ABB RobotStudio station: Estacion_Proyecto.rspag

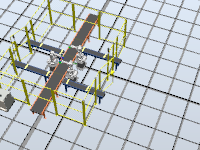
--- station ---
Station Estacion_Proyecto (saved by RobotStudio 20.4.9280.0)
Controller Controlador_Vajilla, task T_ROB3: task frame (RAPID world) sits at (0, 0, 0) mm in the station
Controller Controlador_Vajilla, task T_ROB2: task frame (RAPID world) sits at (0, 0, 0) mm in the station
Controller Controlador_Vajilla, task T_ROB1: task frame (RAPID world) sits at (0, 0, 0) mm in the station
Controller Controlador_Vajilla
  mechanical unit ROB_1: IRB140_6_81_C_03_1, 6 joints, base frame (0, 570, 550) mm, rotated rx 0 ry 0 rz -90 deg
  mechanical unit ROB_2: IRB140_6_81_C_03_2, 6 joints, base frame (1000, 555, 550) mm, rotated rx 0 ry 0 rz -90 deg
  mechanical unit ROB_3: IRB140_6_81_C_03_3, 6 joints, base frame (732.5, -570, 550) mm, rotated rx 0 ry 0 rz 90 deg
Layout (positions relative to the parent item):
  - IRB140_6_81_C_03_1 [mechanism, from Robots\IRB140_6_81_C_G_03.rslib] at (0, 570, 550) mm, rotated rx 0 ry 0 rz -90 deg; joint values [0, 0, 0, 0, 0.5236, 0] (rad or m)
  - IRB140_6_81_C_03_2 [mechanism, from Robots\IRB140_6_81_C_G_03.rslib] at (1000, 555, 550) mm, rotated rx 0 ry 0 rz -90 deg; joint values [0, -0.0417, 0.0409, 0, 0.5244, 0] (rad or m)
  - IRB140_6_81_C_03_3 [mechanism, from Robots\IRB140_6_81_C_G_03.rslib] at (732.5, -570, 550) mm, rotated rx 0 ry 0 rz 90 deg; joint values [0, 0, 0, 0, 0.5236, 0] (rad or m)
  - Sockel_IRB140_500mm_3 [part, from Proyecto\53244bc2-0fdb-48b8-abaf-b031e49cfeeesockel_irb140_500mm.rslib] at (732.5, -570, 0) mm, rotated rx 0 ry 0 rz 90 deg
  - Sockel_IRB140_500mm_1 [part, from Proyecto\53244bc2-0fdb-48b8-abaf-b031e49cfeeesockel_irb140_500mm.rslib] at (0, 570, 0) mm, rotated rx 0 ry 0 rz -90 deg
  - Sockel_IRB140_500mm_2 [part, from Proyecto\53244bc2-0fdb-48b8-abaf-b031e49cfeeesockel_irb140_500mm.rslib] at (1000, 555, 0) mm, rotated rx 0 ry 0 rz -90 deg
  - Linea_Plato_Pando [part] at (-250, 0, 0) mm
  - Linea_Plato_Postre [part] at (0, -6.06, 0) mm
  - Linea_Plato_Hondo [part]
  - Linea_Vaso [part]
  - VacuumToolCreator [smart component, from Proyecto\d28571e4-d633-4a15-b430-832653a4066fvacuumtoolcreator.rslib]
      properties: Tool Name=VacuumTool; TCP Name=tVacuum; TCP Position=[0 0 0.049]; TCP Orientation=[0 0 0]; Flange Diameter=0.055; Length=0.1; Width=0.1; Solids only=false; GeneratedTool=VacuumTool
  - VacuumTool [mechanism, from modelados\VacuumTool.rslib] at (0, 63.71, 1229.5) mm, rotated rx 180 ry 60 rz 90 deg
  - Conveyor_PH [smart component]
      signals: DO ACR, DI ACV, DI DCV, DI INC
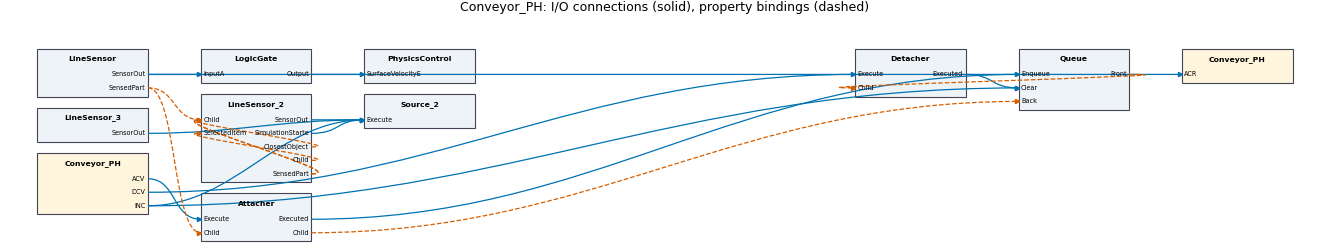
      connections:
        LineSensor.SensorOut -> LogicGate.InputA
        LogicGate.Output -> PhysicsControl.SurfaceVelocityEnabled
        LineSensor_2.SensorOut -> Source_2.Execute
        LineSensor_3.SensorOut -> Source_2.Execute
        SimulationEvents.SimulationStarted -> Source_2.Execute
        LineSensor.SensorOut -> Conveyor_PH.ACR
        Conveyor_PH.ACV -> Attacher.Execute
        Attacher.Executed -> Queue.Enqueue
        Detacher.Executed -> Queue.Clear
        Conveyor_PH.DCV -> Detacher.Execute
        Conveyor_PH.INC -> Source_2.Execute
        Conveyor_PH.INC -> Queue.Clear
        LineSensor.SensedPart => Attacher.Child
        ClosestObject.ClosestObject => Detacher.Child
        Attacher.Child => DataTable.SelectedItem
        VolumeSensor.SensedPart => Detacher.Child
        LineSensor_5.SensedPart => Detacher.Child
        LineSensor.SensedPart => Attacher.Child
        Attacher.Child => Queue.Back
        Queue.Front => Detacher.Child
    - Source_2 [smart component, from Components\Source.rslib] at (159.05, -900.89, 1238.71) mm, rotated rx -56.63 ry -24.63 rz -15.35 deg
        properties: Source=plato_hondo; Copy=(none); Parent=(none); Position=[-0.55 2.2 0.6]; Orientation=[0 0 0]; Transient=true; PhysicsBehavior=3
    - LineSensor [smart component, from Components\LineSensor.rslib]
        properties: Start=[-0.4 0.47 0.6405]; End=[-0.7 0.47 0.6405]; Radius=0.004; SensedPart=(none); SensedPoint=[0 0 0]
      - _sensorPart_ [part]
    - PhysicsControl [smart component, from Components\PhysicsControl.rslib] at (0, -15, 0) mm
        properties: Object=Linea_Plato_Hondo; Behavior=1; SurfaceVelocity=0.3302
    - LogicGate [smart component, from Components\LogicGate.rslib]
        properties: Operator=NOT; Delay=0
    - LineSensor_3 [smart component, from Components\LineSensor.rslib]
        properties: Start=[-0.4 1.6 0.6405]; End=[-0.7 1.6 0.6405]; Radius=0.004; SensedPart=(none); SensedPoint=[0 0 0]
      - _sensorPart_ [part]
    - Attacher [smart component, from Components\Attacher.rslib]
        properties: Parent=VacuumTool; Flange=0; Child=(none); Mount=false; Offset=[0 0 0]; Orientation=[0 0 0]
    - Queue [smart component, from Components\Queue.rslib]
        properties: Back=(none); Front=(none); Queue=; NumberOfObjects=0
    - Detacher [smart component, from Components\Detacher.rslib]
        properties: Child=(none); KeepPosition=true
  - Conveyor_Principal [smart component]
      signals: DI INC, DI MOV, DO ACR_1P, DO ACR_3P
      connections:
        Conveyor_Principal.INC -> Source.Execute
        Conveyor_Principal.MOV -> LogicGate_2.InputA
        LogicGate.Output -> LogicGate_2.InputB
        LogicGate_2.Output -> PhysicsControl.SurfaceVelocityEnabled
        PlaneSensor.SensorOut -> LogicGate.InputA
        PlaneSensor.SensorOut -> Conveyor_Principal.ACR_1P
        PlaneSensor_2.SensorOut -> Conveyor_Principal.ACR_3P
        PlaneSensor_3.SensorOut -> Source.Execute
    - PhysicsControl [smart component, from Components\PhysicsControl.rslib]
        properties: Object=Linea_Principal; Behavior=1; SurfaceVelocity=0.3
    - Source [smart component, from Components\Source.rslib] at (-3.56, 0, 724.94) mm
        properties: Source=caja; Copy=(none); Parent=(none); Position=[-2.5 0 0.6]; Orientation=[0 0 3.14159265358979]; Transient=true; PhysicsBehavior=3
    - LogicGate [smart component, from Components\LogicGate.rslib]
        properties: Operator=NOT; Delay=0
    - LogicGate_2 [smart component, from Components\LogicGate.rslib]
        properties: Operator=OR; Delay=0
    - PlaneSensor [smart component, from Components\PlaneSensor.rslib]
        properties: Origin=[0.12 -0.3 0.605]; Axis1=[0 0.6 0]; Axis2=[0 0 0.1]; SensedPart=(none)
      - _sensorPart_ [part]
    - PlaneSensor_2 [smart component, from Components\PlaneSensor.rslib]
        properties: Origin=[1.3 -0.26 0.605]; Axis1=[-0.00064 0.52 0]; Axis2=[0 0 0.1]; SensedPart=(none)
      - _sensorPart_ [part]
    - PlaneSensor_3 [smart component, from Components\PlaneSensor.rslib]
        properties: Origin=[-1.03 -0.3 0.601]; Axis1=[3E-06 0.6 0]; Axis2=[0 0 0.1]; SensedPart=(none)
      - _sensorPart_ [part]
  - Conveyor_PP [smart component]
      signals: DI ACV_3, DI DCV_3, DI INC_3, DO ACR_3
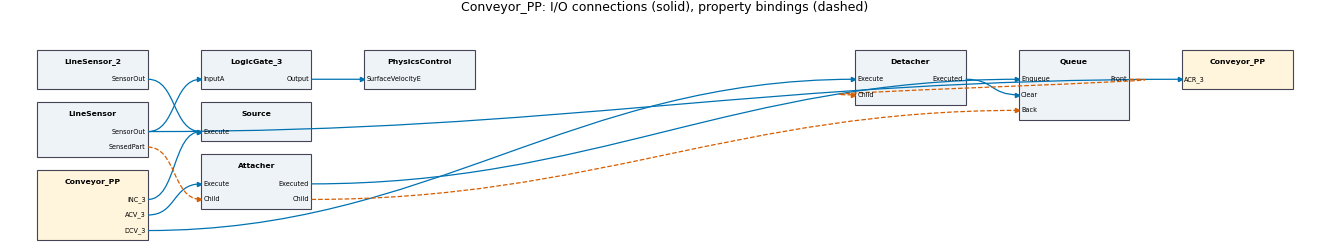
      connections:
        LineSensor_2.SensorOut -> Source.Execute
        LineSensor.SensorOut -> LogicGate_3.InputA
        LogicGate_3.Output -> PhysicsControl.SurfaceVelocityEnabled
        Attacher.Executed -> Queue.Enqueue
        Detacher.Executed -> Queue.Clear
        Conveyor_PP.INC_3 -> Source.Execute
        LineSensor.SensorOut -> Conveyor_PP.ACR_3
        Conveyor_PP.ACV_3 -> Attacher.Execute
        Conveyor_PP.DCV_3 -> Detacher.Execute
        LineSensor.SensedPart => Attacher.Child
        Attacher.Child => Queue.Back
        Queue.Front => Detacher.Child
    - LogicGate_3 [smart component, from Components\LogicGate.rslib]
        properties: Operator=NOT; Delay=0
    - Source [smart component, from Components\Source.rslib]
        properties: Source=plato_pando; Copy=(none); Parent=(none); Position=[0 -2.252 0.601]; Orientation=[0 0 0]; Transient=true; PhysicsBehavior=3
    - PhysicsControl [smart component, from Components\PhysicsControl.rslib]
        properties: Object=Linea_Plato_Pando; Behavior=1; SurfaceVelocity=0.3302
    - LineSensor [smart component, from Components\LineSensor.rslib]
        properties: Start=[-0.15 -0.47 0.615]; End=[0.15 -0.47 0.615]; Radius=0.004; SensedPart=(none); SensedPoint=[0 0 0]
      - _sensorPart_ [part]
    - LineSensor_2 [smart component, from Components\LineSensor.rslib]
        properties: Start=[-0.15 -1.6 0.615]; End=[0.15 -1.6 0.615]; Radius=0.004; SensedPart=(none); SensedPoint=[0 0 0]
      - _sensorPart_ [part]
    - Detacher [smart component, from Components\Detacher.rslib]
        properties: Child=(none); KeepPosition=true
    - Attacher [smart component, from Components\Attacher.rslib]
        properties: Parent=VacuumTool_2; Flange=0; Child=(none); Mount=false; Offset=[0 0 0]; Orientation=[0 0 0]
    - Queue [smart component, from Components\Queue.rslib]
        properties: Back=(none); Front=(none); Queue=; NumberOfObjects=0
  - SimulationEvents [smart component, from Components\SimulationEvents.rslib]
  - VacuumTool_2 [mechanism, from modelados\VacuumTool.rslib] at (732.5, -63.71, 1229.5) mm, rotated rx 180 ry 60 rz -90 deg
  - Conveyor_PPo [smart component]
      signals: DI ACV_3, DI DCV_3, DI INC_3, DO ACR_3
      connections:
        LineSensor_2.SensorOut -> Source.Execute
        LineSensor.SensorOut -> LogicGate.InputA
        LogicGate.Output -> PhysicsControl.SurfaceVelocityEnabled
        Attacher.Executed -> Queue.Enqueue
        Detacher.Executed -> Queue.Clear
        Conveyor_PPo.ACV_3 -> Attacher.Execute
        Conveyor_PPo.DCV_3 -> Detacher.Execute
        Conveyor_PPo.INC_3 -> Source.Execute
        LineSensor.SensorOut -> Conveyor_PPo.ACR_3
        LineSensor.SensedPart => Attacher.Child
        Attacher.Child => Queue.Back
        Queue.Front => Detacher.Child
    - Attacher [smart component, from Components\Attacher.rslib]
        properties: Parent=VacuumTool_2; Flange=0; Child=(none); Mount=false; Offset=[0 0 0]; Orientation=[0 0 0]
    - Detacher [smart component, from Components\Detacher.rslib]
        properties: Child=(none); KeepPosition=true
    - LineSensor [smart component, from Components\LineSensor.rslib]
        properties: Start=[1.315 -0.47 0.615]; End=[1.615 -0.47 0.615]; Radius=0.004; SensedPart=(none); SensedPoint=[0 0 0]
      - _sensorPart_ [part]
    - LineSensor_2 [smart component, from Components\LineSensor.rslib]
        properties: Start=[1.315 -1.6 0.618]; End=[1.615 -1.6 0.618]; Radius=0.004; SensedPart=(none); SensedPoint=[0 0 0]
      - _sensorPart_ [part]
    - PhysicsControl [smart component, from Components\PhysicsControl.rslib]
        properties: Object=Linea_Plato_Postre; Behavior=1; SurfaceVelocity=0.3302
    - Queue [smart component, from Components\Queue.rslib]
        properties: Back=(none); Front=(none); Queue={24e2353d-62ec-438d-8f5e-047144dff703}; NumberOfObjects=1
    - Source [smart component, from Components\Source.rslib]
        properties: Source=plato_postre; Copy=(none); Parent=(none); Position=[1.465 -2.252 0.601]; Orientation=[0 0 0]; Transient=true; PhysicsBehavior=3
    - LogicGate [smart component, from Components\LogicGate.rslib]
        properties: Operator=NOT; Delay=0
  - LogicGate [smart component, from Components\LogicGate.rslib]
      properties: Operator=AND; Delay=0
  - plato_postre [part]
  - plato_pando [part]
  - plato_hondo [part]
  - VacuumTool1x1 [mechanism, from modelados\VacuumTool1x1.rslib] at (1000, 63.71, 1229.5) mm, rotated rx -180 ry 60 rz 90 deg
  - Conveyor_V [smart component]
      signals: DI ACV_2, DI DCV_2, DI INC_2, DO ACV_R2
      connections:
        LineSensor_3.SensorOut -> LogicGate.InputA
        LogicGate.Output -> PhysicsControl.SurfaceVelocityEnabled
        LineSensor_4.SensorOut -> Source.Execute
        Attacher.Executed -> Queue.Enqueue
        Detacher.Executed -> Queue.Clear
        Conveyor_V.ACV_2 -> Attacher.Execute
        Conveyor_V.DCV_2 -> Detacher.Execute
        Conveyor_V.INC_2 -> Source.Execute
        LineSensor_3.SensorOut -> Conveyor_V.ACV_R2
        LineSensor_3.SensedPart => Attacher.Child
        Attacher.Child => Queue.Back
        Queue.Front => Detacher.Child
    - Attacher [smart component, from Components\Attacher.rslib]
        properties: Parent=VacuumTool1x1; Flange=0; Child=(none); Mount=false; Offset=[0 0 0]; Orientation=[0 0 0]
    - Detacher [smart component, from Components\Detacher.rslib]
        properties: Child=(none); KeepPosition=true
    - LineSensor_3 [smart component, from Components\LineSensor.rslib]
        properties: Start=[1.7 0.6 0.6405]; End=[1.4 0.6 0.6405]; Radius=0.004; SensedPart=(none); SensedPoint=[0 0 0]
      - _sensorPart_ [part]
    - LineSensor_4 [smart component, from Components\LineSensor.rslib]
        properties: Start=[1.7 1.6 0.6405]; End=[1.4 1.6 0.6405]; Radius=0.004; SensedPart=(none); SensedPoint=[0 0 0]
      - _sensorPart_ [part]
    - PhysicsControl [smart component, from Components\PhysicsControl.rslib]
        properties: Object=Linea_Vaso; Behavior=1; SurfaceVelocity=0.2
    - Queue [smart component, from Components\Queue.rslib]
        properties: Back=(none); Front=(none); Queue=; NumberOfObjects=0
    - Source [smart component, from Components\Source.rslib] at (-390.95, 83.44, -137.11) mm, rotated rx 0 ry 0 rz -28.76 deg
        properties: Source=vaso; Copy=(none); Parent=(none); Position=[1.55 2.2 0.711]; Orientation=[3.14159265358979 0 0]; Transient=true; PhysicsBehavior=3
    - LogicGate [smart component, from Components\LogicGate.rslib]
        properties: Operator=NOT; Delay=0
  - vaso [part]
  - Fence [graphiccomponentgroup]
    - Segment 1 [part]
    - Segment 2 [part]
    - Segment 3 [part]
    - Segment 4 [part]
    - Segment 5 [part]
    - Segment 6 [part]
  - Fence [graphiccomponentgroup]
    - Segment 7 [part]
    - Segment 8 [part]
    - Segment 9 [part]
  - Fence [graphiccomponentgroup]
    - Segment 1 [part]
    - Segment 2 [part]
    - Segment 3 [part]
    - Segment 4 [part]
    - Segment 5 [part]
    - Segment 6 [part]
    - Segment 7 [part]
  - Fence [graphiccomponentgroup]
    - Segment 1 [part]
    - Segment 2 [part]
    - Segment 3 [part]
    - Segment 4 [part]
  - IRC5_Singel-Cabinet [part, from Equipment\IRC5_Singel-Cabinet.rslib] at (3600, -1753.51, 100) mm, rotated rx 90 ry 0 rz 90 deg
  - FlexPendant [part, from Equipment\FlexPendant.rslib] at (3600, -1753.51, 1000) mm, rotated rx -30 ry 0 rz 90 deg
  - Part_2 [part]
  - Linea_Principal [part]
  - caja [part] at (0, -3099.64, 0) mm
  - SC_StatusLamps [smart component, from modelados\6343e143-9244-4892-8935-83fad9482edbsc_statuslamps.rslib] at (1233.15, -2105.74, 2000) mm
      properties: OK=green; Warning=yellow; Error=red
    - warning lamps [part, from modelados\6343e143-9244-4892-8935-83fad9482edbsc_statuslamps.rslib]
    - green [part, from modelados\6343e143-9244-4892-8935-83fad9482edbsc_statuslamps.rslib] at (102.3, 1404.98, -880.75) mm
    - yellow [part, from modelados\6343e143-9244-4892-8935-83fad9482edbsc_statuslamps.rslib] at (102.3, 1404.98, -880.75) mm
    - red [part, from modelados\6343e143-9244-4892-8935-83fad9482edbsc_statuslamps.rslib] at (102.3, 1404.98, -880.75) mm
  - LogicGate_2 [smart component, from Components\LogicGate.rslib]
      properties: Operator=OR; Delay=0
  - LogicGate_3 [smart component, from Components\LogicGate.rslib]
      properties: Operator=OR; Delay=0
  - LogicGate_4 [smart component, from Components\LogicGate.rslib]
      properties: Operator=OR; Delay=0
  - LogicGate_5 [smart component, from Components\LogicGate.rslib]
      properties: Operator=OR; Delay=0
  - SC_StatusLamps_2 [smart component, from modelados\6343e143-9244-4892-8935-83fad9482edbsc_statuslamps.rslib] at (317.5, 2100, 2000) mm
      properties: OK=green; Warning=yellow; Error=red
    - warning lamps [part, from modelados\6343e143-9244-4892-8935-83fad9482edbsc_statuslamps.rslib]
    - green [part, from modelados\6343e143-9244-4892-8935-83fad9482edbsc_statuslamps.rslib] at (102.3, 1404.98, -880.75) mm
    - yellow [part, from modelados\6343e143-9244-4892-8935-83fad9482edbsc_statuslamps.rslib] at (102.3, 1404.98, -880.75) mm
    - red [part, from modelados\6343e143-9244-4892-8935-83fad9482edbsc_statuslamps.rslib] at (102.3, 1404.98, -880.75) mm
Attachment: Source_2 is attached to IRB140_6_81_C_03_1 / Link6
Attachment: PhysicsControl is attached to Sockel_IRB140_500mm_2
Attachment: Sockel_IRB140_500mm_3 is attached to IRB140_6_81_C_03_3 / Base
Attachment: Sockel_IRB140_500mm_1 is attached to IRB140_6_81_C_03_1 / Base
Attachment: Sockel_IRB140_500mm_2 is attached to IRB140_6_81_C_03_2 / Base
Attachment: VacuumTool is attached to IRB140_6_81_C_03_1 / Link6
Attachment: VacuumTool_2 is attached to IRB140_6_81_C_03_3 / Link6
Attachment: VacuumTool1x1 is attached to IRB140_6_81_C_03_2 / Link6
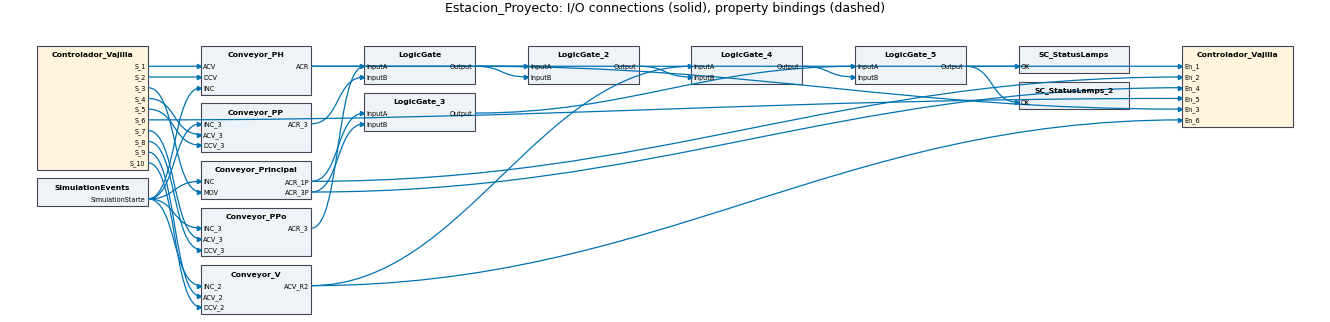
Station logic (signal -> signal, property => property):
  Conveyor_PH.ACR -> Controlador_Vajilla.En_1
  Controlador_Vajilla.S_1 -> Conveyor_PH.ACV
  Controlador_Vajilla.S_2 -> Conveyor_PH.DCV
  SimulationEvents.SimulationStarted -> Conveyor_PH.INC
  SimulationEvents.SimulationStarted -> Conveyor_Principal.INC
  Controlador_Vajilla.S_3 -> Conveyor_Principal.MOV
  Conveyor_Principal.ACR_1P -> Controlador_Vajilla.En_2
  SimulationEvents.SimulationStarted -> Conveyor_PP.INC_3
  Controlador_Vajilla.S_4 -> Conveyor_PP.ACV_3
  Controlador_Vajilla.S_5 -> Conveyor_PP.DCV_3
  Conveyor_Principal.ACR_3P -> Controlador_Vajilla.En_4
  Controlador_Vajilla.S_6 -> Controlador_Vajilla.En_5
  SimulationEvents.SimulationStarted -> Conveyor_PPo.INC_3
  Controlador_Vajilla.S_7 -> Conveyor_PPo.ACV_3
  Controlador_Vajilla.S_8 -> Conveyor_PPo.DCV_3
  Conveyor_PPo.ACR_3 -> LogicGate.InputA
  Conveyor_PP.ACR_3 -> LogicGate.InputB
  LogicGate.Output -> Controlador_Vajilla.En_3
  SimulationEvents.SimulationStarted -> Conveyor_V.INC_2
  Controlador_Vajilla.S_9 -> Conveyor_V.ACV_2
  Controlador_Vajilla.S_10 -> Conveyor_V.DCV_2
  Conveyor_V.ACV_R2 -> Controlador_Vajilla.En_6
  Conveyor_PH.ACR -> LogicGate_2.InputA
  LogicGate.Output -> LogicGate_2.InputB
  Conveyor_Principal.ACR_1P -> LogicGate_3.InputA
  Conveyor_Principal.ACR_3P -> LogicGate_3.InputB
  Conveyor_V.ACV_R2 -> LogicGate_4.InputA
  LogicGate_2.Output -> LogicGate_4.InputB
  LogicGate_3.Output -> LogicGate_5.InputA
  LogicGate_4.Output -> LogicGate_5.InputB
  LogicGate_5.Output -> SC_StatusLamps.OK
  LogicGate_5.Output -> SC_StatusLamps_2.OK

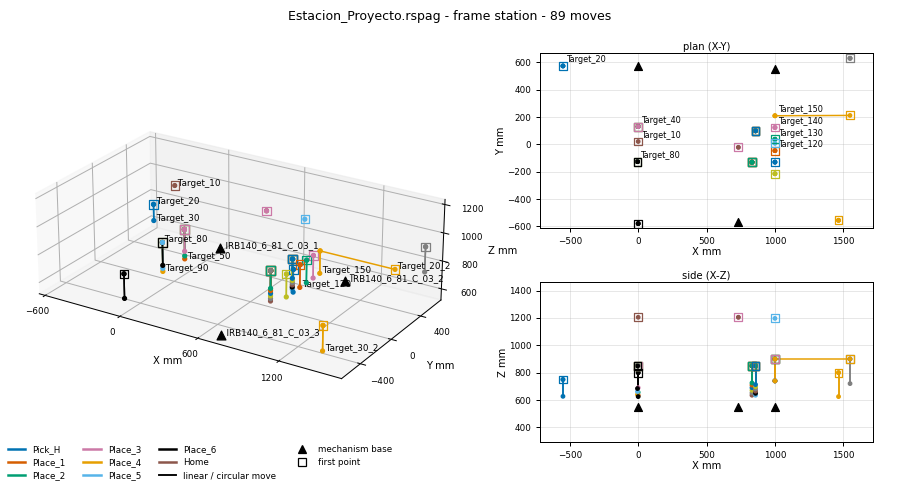
[picture p0: tool path of Estacion_Proyecto.rspag in frame station, 89 of 89 moves have a stored position in this frame; points joined in program order, loops and branches not executed]
--- Backups/Controlador_Vajilla/RAPID/TASK1/PROGMOD/CalibData.mod ---
MODULE CalibData
    PERS tooldata tVacuum:=[TRUE,[[0,0,49],[1,0,0,0]],[1,[0,0,32.6667],[1,0,0,0],0,0,0]];
    TASK PERS wobjdata PlatoH:=[FALSE,TRUE,"",[[-550,400,600],[1,0,0,0]],[[0,0,0],[1,0,0,0]]];
    TASK PERS wobjdata Principal:=[FALSE,TRUE,"",[[-2000,0,600],[1,0,0,0]],[[0,0,0],[1,0,0,0]]];
ENDMODULE

--- Backups/Controlador_Vajilla/RAPID/TASK1/PROGMOD/Module1.mod ---
MODULE Module1
    CONST robtarget Target_10:=[[550,-378.726896031,605],[0.353553391,0.612372436,0.612372436,-0.353553391],[0,0,0,0],[9E+09,9E+09,9E+09,9E+09,9E+09,9E+09]];
    CONST robtarget Target_20:=[[0,173.72,150],[0,0.707106781,0.707106781,0],[-2,0,-2,0],[9E+09,9E+09,9E+09,9E+09,9E+09,9E+09]];
    CONST robtarget Target_30:=[[0,173.72,27],[0,0.707106781,0.707106781,0],[-2,-1,-2,0],[9E+09,9E+09,9E+09,9E+09,9E+09,9E+09]];
    CONST robtarget Target_40:=[[2000,130.5,250],[0,0,1,0],[0,-1,-2,0],[9E+09,9E+09,9E+09,9E+09,9E+09,9E+09]];
    CONST robtarget Target_50:=[[2000,130.5,34],[0,0,1,0],[0,-1,-2,0],[9E+09,9E+09,9E+09,9E+09,9E+09,9E+09]];
    CONST robtarget Target_60:=[[2000,130.5,56],[0,0,1,0],[-1,0,-2,0],[9E+09,9E+09,9E+09,9E+09,9E+09,9E+09]];
    CONST robtarget Target_70:=[[2000,130.5,90],[0,0,1,0],[0,-1,-2,0],[9E+09,9E+09,9E+09,9E+09,9E+09,9E+09]];
    CONST robtarget Target_80:=[[1995,-126,250],[0,0,1,0],[0,-1,-2,0],[9E+09,9E+09,9E+09,9E+09,9E+09,9E+09]];
    CONST robtarget Target_90:=[[1995,-126,40],[0,0,1,0],[0,0,-2,0],[9E+09,9E+09,9E+09,9E+09,9E+09,9E+09]];
    CONST robtarget Target_100:=[[1995,-126,62],[0,0,1,0],[0,0,-2,0],[9E+09,9E+09,9E+09,9E+09,9E+09,9E+09]];
    CONST robtarget Target_110:=[[1995,-126,84],[0,0,1,0],[0,0,-2,0],[9E+09,9E+09,9E+09,9E+09,9E+09,9E+09]];
    VAR num i;


    !***********************************************************
    !
    ! Module:  Module1
    !
    ! Description:
    !   <Insert description here>
    !
    ! Author: santi
    !
    ! Version: 1.0
    !
    !***********************************************************


    !***********************************************************
    !
    ! Procedure main
    !
    !   This is the entry point of your program
    !
    !***********************************************************
    PROC main()
        !Add your code here
        Home;
        i:=1;

        WHILE i<=6 DO
            WaitDI En_1,1;
            WaitDI En_2,1;
            Pick_H;
            IF i=1 THEN
                Place_1;
                Incr i;
            ELSEIF i=2 THEN

                Place_2;
                Incr i;
            ELSEIF i=3 THEN

                Place_3;
                Incr i;
            ELSEIF i=4 THEN

                Place_4;
                Incr i;
            ELSEIF i=5 THEN

                Place_5;
                Incr i;
            ELSEIF i=6 THEN

                Place_6;
                WaitDI En_5,1;
                SetDO S_3,1;
                WaitDI En_2,0;
                WaitDI En_2,1;
                SetDO S_3,0;
                i:=1;
            ENDIF
        ENDWHILE


        !        Pick_H;
        !        Place_1;
        !        Pick_H;
        !        Place_2;
        !        Pick_H;
        !        Place_3;
        !        Pick_H;
        !        Place_4;
        !        Pick_H;
        !        Place_5;
        !        Pick_H;
        !        Place_6;

    ENDPROC

    PROC Pick_H()
        MoveJ Target_20,v2500,z10,tVacuum\WObj:=PlatoH;
        MoveL Target_30,v300,fine,tVacuum\WObj:=PlatoH;
        SetDO S_1,1;
        WaitTime 1;
        SetDO S_1,0;
        MoveL Target_20,v300,z10,tVacuum\WObj:=PlatoH;
    ENDPROC

    PROC Place_1()
        MoveL Target_40,v2000,z10,tVacuum\WObj:=Principal;
        MoveL Target_50,v300,fine,tVacuum\WObj:=Principal;
        SetDO S_2,1;
        SetDO S_2,0;
        MoveL Target_40,v2000,z10,tVacuum\WObj:=Principal;
    ENDPROC

    PROC Place_2()
        MoveL Target_40,v2000,z10,tVacuum\WObj:=Principal;
        MoveL Target_60,v300,fine,tVacuum\WObj:=Principal;
        SetDO S_2,1;
        SetDO S_2,0;
        MoveL Target_40,v2000,z10,tVacuum\WObj:=Principal;
    ENDPROC

    PROC Place_3()
        MoveL Target_40,v2000,z10,tVacuum\WObj:=Principal;
        MoveL Target_70,v300,fine,tVacuum\WObj:=Principal;
        SetDO S_2,1;
        SetDO S_2,0;
        MoveL Target_40,v2000,z10,tVacuum\WObj:=Principal;
    ENDPROC

    PROC Place_4()
        MoveL Target_80,v2000,z10,tVacuum\WObj:=Principal;
        MoveL Target_90,v300,fine,tVacuum\WObj:=Principal;
        SetDO S_2,1;
        SetDO S_2,0;
        MoveL Target_80,v2000,z10,tVacuum\WObj:=Principal;
    ENDPROC

    PROC Place_5()
        MoveL Target_80,v2000,z10,tVacuum\WObj:=Principal;
        MoveL Target_100,v300,fine,tVacuum\WObj:=Principal;
        SetDO S_2,1;
        SetDO S_2,0;
        MoveL Target_80,v2000,z10,tVacuum\WObj:=Principal;
    ENDPROC

    PROC Place_6()
        MoveL Target_80,v2000,z10,tVacuum\WObj:=Principal;
        MoveL Target_110,v300,fine,tVacuum\WObj:=Principal;
        SetDO S_2,1;
        SetDO S_2,0;
        MoveL Target_80,v2000,z10,tVacuum\WObj:=Principal;
        Home;
    ENDPROC

    PROC Home()
        MoveJ Target_10,v2500,z1,tVacuum\WObj:=PlatoH;
    ENDPROC
ENDMODULE

--- Backups/Controlador_Vajilla/RAPID/TASK2/PROGMOD/CalibData.mod ---
MODULE CalibData
    PERS tooldata MyTool:=[TRUE,[[31.7926,0,229.639],[0.945519,0,0.325568,0]],[1,[0,0,1],[1,0,0,0],0,0,0]];
    PERS tooldata wrist0:=[TRUE,[[0,0,129],[1,0,0,0]],[1,[0,0,100],[1,0,0,0],0,0,0]];
    PERS tooldata VacuumTool1x1:=[TRUE,[[0,0,65],[1,0,0,0]],[0.2,[0,0,1],[1,0,0,0],0,0,0]];
    TASK PERS wobjdata Vaso:=[FALSE,TRUE,"",[[1550,400,600],[1,0,0,0]],[[0,0,0],[1,0,0,0]]];
    TASK PERS wobjdata Principal:=[FALSE,TRUE,"",[[-2000,0,600],[1,0,0,0]],[[0,0,0],[1,0,0,0]]];
ENDMODULE

--- Backups/Controlador_Vajilla/RAPID/TASK2/PROGMOD/Module1.mod ---
MODULE Module1
        CONST robtarget Target_20:=[[-1,229.65,300],[0,0.707106781,0.707106781,0],[0,0,0,0],[9E+09,9E+09,9E+09,9E+09,9E+09,9E+09]];
    CONST robtarget Target_30:=[[-1,229.62,120],[0,0.707106781,0.707106781,0],[0,0,0,0],[9E+09,9E+09,9E+09,9E+09,9E+09,9E+09]];
    CONST robtarget Target_40:=[[3000,-214.5,300],[0,0.707106781,0.707106781,0],[0,0,0,0],[9E+09,9E+09,9E+09,9E+09,9E+09,9E+09]];
    CONST robtarget Target_100:=[[3000,-214.5,140],[0,0.707106781,0.707106781,0],[0,0,0,0],[9E+09,9E+09,9E+09,9E+09,9E+09,9E+09]];
    CONST robtarget Target_50:=[[3000,-129.5,300],[0,0.707106781,0.707106781,0],[0,-1,0,0],[9E+09,9E+09,9E+09,9E+09,9E+09,9E+09]];
    CONST robtarget Target_110:=[[3000,-129.5,140],[0,0.707106781,0.707106781,0],[0,-1,0,0],[9E+09,9E+09,9E+09,9E+09,9E+09,9E+09]];
    CONST robtarget Target_60:=[[3000,-45.5,300],[0,0.707106781,0.707106781,0],[0,-1,0,0],[9E+09,9E+09,9E+09,9E+09,9E+09,9E+09]];
    CONST robtarget Target_120:=[[3000,-45.5,140],[0,0.707106781,0.707106781,0],[0,-1,0,0],[9E+09,9E+09,9E+09,9E+09,9E+09,9E+09]];
    CONST robtarget Target_70:=[[3000,37.5,300],[0,0.707106781,0.707106781,0],[0,0,0,0],[9E+09,9E+09,9E+09,9E+09,9E+09,9E+09]];
    CONST robtarget Target_130:=[[3000,37.5,140],[0,0.707106781,0.707106781,0],[0,0,0,0],[9E+09,9E+09,9E+09,9E+09,9E+09,9E+09]];
    CONST robtarget Target_80:=[[3000,123.5,300],[0,0.707106781,0.707106781,0],[0,-1,0,0],[9E+09,9E+09,9E+09,9E+09,9E+09,9E+09]];
    CONST robtarget Target_140:=[[3000,123.5,140],[0,0.707106781,0.707106781,0],[0,-1,0,0],[9E+09,9E+09,9E+09,9E+09,9E+09,9E+09]];
    CONST robtarget Target_90:=[[3000,209.5,300],[0,0.707106781,0.707106781,0],[0,-1,0,0],[9E+09,9E+09,9E+09,9E+09,9E+09,9E+09]];
    CONST robtarget Target_150:=[[3000,209.5,140],[0,0.707106781,0.707106781,0],[0,-1,0,0],[9E+09,9E+09,9E+09,9E+09,9E+09,9E+09]];
    CONST robtarget Target_10:=[[-550,-392.583302492,597],[0.353553391,0.612372436,0.612372436,-0.353553391],[0,0,0,0],[9E+09,9E+09,9E+09,9E+09,9E+09,9E+09]];
    CONST robtarget Target_20_2:=[[-1.46,-188,300],[0,0.707106781,0.707106781,0],[0,0,0,0],[9E+09,9E+09,9E+09,9E+09,9E+09,9E+09]];
!***********************************************************
    !
    ! Module:  Module1
    !
    ! Description:
    !   <Insert description here>
    !
    ! Author: santi
    !
    ! Version: 1.0
    !
    !***********************************************************


    !***********************************************************
    !
    ! Procedure main
    !
    !   This is the entry point of your program
    !
    !***********************************************************
    PROC main()
        !Add your code here

        Home_V;
        Proceso_R2:
        WaitDI En_6,1;
        WaitDI En_4,1;
        Pick_V;
        Place_1_V;
        Pick_V;
        Place_2_V;
        Pick_V;
        Place_3_V;
        Pick_V;
        Place_4_V;
        Pick_V;
        Place_5_V;
        Pick_V;
        Place_6_V;
        WaitDI En_4,0;
        GOTO Proceso_R2;
    ENDPROC
    PROC Pick_V()
        MoveJ Target_20,v2000,z10,VacuumTool1x1\WObj:=Vaso;
        MoveL Target_30,v300,fine,VacuumTool1x1\WObj:=Vaso;
        SetDO S_9,1;
        WaitTime 1;
        SetDO S_9,0;
        MoveL Target_20,v300,z10,VacuumTool1x1\WObj:=Vaso;
    ENDPROC
    PROC Place_1_V()
        MoveL Target_40,v1000,z10,VacuumTool1x1\WObj:=Principal;
        MoveL Target_100,v200,fine,VacuumTool1x1\WObj:=Principal;
        SetDO S_10,1;
        SetDO S_10,0;
        MoveL Target_40,v1000,z10,VacuumTool1x1\WObj:=Principal;
    ENDPROC
    PROC Place_2_V()
        MoveL Target_50,v1000,z10,VacuumTool1x1\WObj:=Principal;
        MoveL Target_110,v200,fine,VacuumTool1x1\WObj:=Principal;
        SetDO S_10,1;
        SetDO S_10,0;
        MoveL Target_50,v1000,z10,VacuumTool1x1\WObj:=Principal;
    ENDPROC
    PROC Place_3_V()
        MoveL Target_60,v1000,z10,VacuumTool1x1\WObj:=Principal;
        MoveL Target_120,v200,fine,VacuumTool1x1\WObj:=Principal;
        SetDO S_10,1;
        SetDO S_10,0;
        MoveL Target_60,v1000,z10,VacuumTool1x1\WObj:=Principal;
    ENDPROC
    PROC Place_4_V()
        MoveL Target_70,v1000,z10,VacuumTool1x1\WObj:=Principal;
        MoveL Target_130,v200,fine,VacuumTool1x1\WObj:=Principal;
        SetDO S_10,1;
        SetDO S_10,0;
        MoveL Target_70,v1000,z10,VacuumTool1x1\WObj:=Principal;
    ENDPROC
    PROC Place_5_V()
        MoveL Target_80,v1000,z10,VacuumTool1x1\WObj:=Principal;
        MoveL Target_140,v200,fine,VacuumTool1x1\WObj:=Principal;
        SetDO S_10,1;
        SetDO S_10,0;
        MoveL Target_80,v1000,z10,VacuumTool1x1\WObj:=Principal;
    ENDPROC
    PROC Place_6_V()
        MoveL Target_20_2,v1000,z10,VacuumTool1x1\WObj:=Vaso;
        MoveL Target_90,v1000,z10,VacuumTool1x1\WObj:=Principal;
        MoveL Target_150,v200,fine,VacuumTool1x1\WObj:=Principal;
        SetDO S_10,1;
        SetDO S_10,0;
        MoveL Target_90,v1000,z10,VacuumTool1x1\WObj:=Principal;
        Home_v;
    ENDPROC
    PROC Home_v()
        MoveJ Target_10,v2000,z10,VacuumTool1x1\WObj:=Vaso;
    ENDPROC
ENDMODULE

--- Backups/Controlador_Vajilla/RAPID/TASK3/PROGMOD/CalibData.mod ---
MODULE CalibData
    PERS tooldata tVacuum:=[TRUE,[[0,0,49],[1,0,0,0]],[1,[0,0,32.6667],[1,0,0,0],0,0,0]];
    TASK PERS wobjdata Plato_P:=[FALSE,TRUE,"",[[0,-400,600],[0,0,0,1]],[[0,0,0],[1,0,0,0]]];
    TASK PERS wobjdata Principal:=[FALSE,TRUE,"",[[-2000,0,600],[1,0,0,0]],[[0,0,0],[1,0,0,0]]];
    TASK PERS wobjdata Plato_Po:=[FALSE,TRUE,"",[[1465,-406.06,600],[0,0,0,1]],[[0,0,0],[1,0,0,0]]];
ENDMODULE

--- Backups/Controlador_Vajilla/RAPID/TASK3/PROGMOD/Module1.mod ---
MODULE Module1
    CONST robtarget Target_20:=[[0,178.82,200],[0,0.707106781,0.707106781,0],[1,0,1,0],[9E+09,9E+09,9E+09,9E+09,9E+09,9E+09]];
    CONST robtarget Target_30:=[[0,178.82,25],[0,0.707106781,0.707106781,0],[1,-1,1,0],[9E+09,9E+09,9E+09,9E+09,9E+09,9E+09]];
    CONST robtarget Target_40:=[[2832,-130,250],[0,0,1,0],[0,0,1,0],[9E+09,9E+09,9E+09,9E+09,9E+09,9E+09]];
    CONST robtarget Target_50:=[[2832,-130,35],[0,0,1,0],[0,0,1,0],[9E+09,9E+09,9E+09,9E+09,9E+09,9E+09]];
    CONST robtarget Target_60:=[[2832,-130,52],[0,0,1,0],[0,-1,1,0],[9E+09,9E+09,9E+09,9E+09,9E+09,9E+09]];
    CONST robtarget Target_70:=[[2832,-130,71],[0,0,1,0],[0,0,1,0],[9E+09,9E+09,9E+09,9E+09,9E+09,9E+09]];
    CONST robtarget Target_80:=[[2832,-130,90],[0,0,1,0],[0,0,1,0],[9E+09,9E+09,9E+09,9E+09,9E+09,9E+09]];
    CONST robtarget Target_90:=[[2832,-130,109],[0,0,1,0],[0,0,1,0],[9E+09,9E+09,9E+09,9E+09,9E+09,9E+09]];
    CONST robtarget Target_100:=[[2832,-130,125],[0,0,1,0],[0,0,1,0],[9E+09,9E+09,9E+09,9E+09,9E+09,9E+09]];

    CONST robtarget Target_20_2:=[[0,148.85,200],[0,0.707106781,0.707106781,0],[-1,0,-1,0],[9E+09,9E+09,9E+09,9E+09,9E+09,9E+09]];
    CONST robtarget Target_30_2:=[[0,148.85,25],[0,0.707106781,0.707106781,0],[-1,0,-1,0],[9E+09,9E+09,9E+09,9E+09,9E+09,9E+09]];
    CONST robtarget Target_110:=[[2857.999998306,100.000014995,249.999986159],[0,-0.000000021,1,0.000000008],[0,-1,1,0],[9E+09,9E+09,9E+09,9E+09,9E+09,9E+09]];
    CONST robtarget Target_120:=[[2857.99999831,100.000014934,35.000017337],[0,-0.000000021,1,0.000000008],[0,-1,1,0],[9E+09,9E+09,9E+09,9E+09,9E+09,9E+09]];
    CONST robtarget Target_130:=[[2857.999999048,99.999999433,48.99996454],[0.000000001,-0.000000021,1,-0.000000022],[0,0,1,0],[9E+09,9E+09,9E+09,9E+09,9E+09,9E+09]];
    CONST robtarget Target_140:=[[2857.999999362,99.999993101,64.999952464],[0.000000002,-0.000000021,1,-0.000000037],[0,-1,1,0],[9E+09,9E+09,9E+09,9E+09,9E+09,9E+09]];
    CONST robtarget Target_150:=[[2858,100,81],[0,0,1,0],[0,0,1,0],[9E+09,9E+09,9E+09,9E+09,9E+09,9E+09]];
    CONST robtarget Target_160:=[[2858,100,97],[0,0,1,0],[0,-1,1,0],[9E+09,9E+09,9E+09,9E+09,9E+09,9E+09]];
    CONST robtarget Target_170:=[[2858,100,113],[0,0,1,0],[0,-1,1,0],[9E+09,9E+09,9E+09,9E+09,9E+09,9E+09]];
    CONST robtarget Target_10:=[[-732.5,-378.726981985,604.999954426],[0.353553387,0.612372438,0.612372438,-0.353553387],[0,0,0,0],[9E+09,9E+09,9E+09,9E+09,9E+09,9E+09]];
    !***********************************************************
    !
    ! Module:  Module1
    !
    ! Description:
    !   <Insert description here>
    !
    ! Author: santi
    !
    ! Version: 1.0
    !
    !***********************************************************


    !***********************************************************
    !
    ! Procedure main
    !
    !   This is the entry point of your program
    !
    !***********************************************************
    PROC main()
        !Add your code here

        Home_R3;
        SetDO S_6,1;
        Proceso_R3:
        WaitDI En_3,1;
        WaitDI En_4,1;
        SetDO S_6,0;
        Pick_PP;
        Place_1_PP;
        Pick_PP;
        Place_2_PP;
        Pick_PP;
        Place_3_PP;
        Pick_PP;
        Place_4_PP;
        Pick_PP;
        Place_5_PP;
        Pick_PP;
        Place_6_PP;

        Pick_PPo;
        Place_1_PPo;
        Pick_PPo;
        Place_2_PPo;
        Pick_PPo;
        Place_3_PPo;
        Pick_PPo;
        Place_4_PPo;
        Pick_PPo;
        Place_5_PPo;
        Pick_PPo;
        Place_6_PPo;
        SetDO S_6,1;
        WaitDI En_4,0;
        GOTO Proceso_R3;
    ENDPROC

    PROC Pick_PP()
        MoveJ Target_20,v2500,z10,tVacuum\WObj:=Plato_P;
        MoveL Target_30,v300,fine,tVacuum\WObj:=Plato_P;
        SetDO S_4,1;
        WaitTime 1;
        SetDO S_4,0;
        MoveL Target_20,v300,z10,tVacuum\WObj:=Plato_P;
    ENDPROC

    PROC Place_1_PP()
        MoveL Target_40,v2000,z10,tVacuum\WObj:=Principal;
        MoveL Target_50,v300,fine,tVacuum\WObj:=Principal;
        SetDO S_5,1;
        SetDO S_5,0;
        MoveL Target_40,v2000,z10,tVacuum\WObj:=Principal;
    ENDPROC

    PROC Place_2_PP()
        MoveL Target_40,v2000,z10,tVacuum\WObj:=Principal;
        MoveL Target_60,v300,fine,tVacuum\WObj:=Principal;
        SetDO S_5,1;
        SetDO S_5,0;
        MoveL Target_40,v2000,z10,tVacuum\WObj:=Principal;
    ENDPROC

    PROC Place_3_PP()
        MoveL Target_40,v2000,z10,tVacuum\WObj:=Principal;
        MoveL Target_70,v300,fine,tVacuum\WObj:=Principal;
        SetDO S_5,1;
        SetDO S_5,0;
        MoveL Target_40,v2000,z10,tVacuum\WObj:=Principal;
    ENDPROC

    PROC Place_4_PP()
        MoveL Target_40,v2000,z10,tVacuum\WObj:=Principal;
        MoveL Target_80,v300,fine,tVacuum\WObj:=Principal;
        SetDO S_5,1;
        SetDO S_5,0;
        MoveL Target_40,v2000,z10,tVacuum\WObj:=Principal;
    ENDPROC

    PROC Place_5_PP()
        MoveL Target_40,v2000,z10,tVacuum\WObj:=Principal;
        MoveL Target_90,v300,fine,tVacuum\WObj:=Principal;
        SetDO S_5,1;
        SetDO S_5,0;
        MoveL Target_40,v2000,z10,tVacuum\WObj:=Principal;
    ENDPROC

    PROC Place_6_PP()
        MoveL Target_40,v2000,z10,tVacuum\WObj:=Principal;
        MoveL Target_100,v300,fine,tVacuum\WObj:=Principal;
        SetDO S_5,1;
        SetDO S_5,0;
        MoveL Target_40,v2000,z10,tVacuum\WObj:=Principal;
        Home_R3;
    ENDPROC

    PROC Home_R3()
        MoveJ Target_10,v2500,z1,tVacuum\WObj:=Plato_P;
    ENDPROC

    PROC Pick_PPo()
        MoveJ Target_20_2,v2500,z10,tVacuum\WObj:=Plato_Po;
        MoveL Target_30_2,v300,fine,tVacuum\WObj:=Plato_Po;
        SetDO S_7,1;
        WaitTime 1;
        SetDO S_7,0;
        MoveL Target_20_2,v300,z10,tVacuum\WObj:=Plato_Po;
    ENDPROC

    PROC Place_1_PPo()
        MoveL Target_110,v2000,z10,tVacuum\WObj:=Principal;
        MoveL Target_120,v300,fine,tVacuum\WObj:=Principal;
        SetDO S_8,1;
        SetDO S_8,0;
        MoveL Target_110,v2000,fine,tVacuum\WObj:=Principal;
    ENDPROC

    PROC Place_2_PPo()
        MoveL Target_110,v2000,z10,tVacuum\WObj:=Principal;
        MoveL Target_130,v300,fine,tVacuum\WObj:=Principal;
        SetDO S_8,1;
        SetDO S_8,0;
        MoveL Target_110,v2000,fine,tVacuum\WObj:=Principal;
    ENDPROC

    PROC Place_3_PPo()
        MoveL Target_110,v2000,z10,tVacuum\WObj:=Principal;
        MoveL Target_140,v300,fine,tVacuum\WObj:=Principal;
        SetDO S_8,1;
        SetDO S_8,0;
        MoveL Target_110,v2000,fine,tVacuum\WObj:=Principal;
    ENDPROC

    PROC Place_4_PPo()
        MoveL Target_110,v2000,z10,tVacuum\WObj:=Principal;
        MoveL Target_150,v300,fine,tVacuum\WObj:=Principal;
        SetDO S_8,1;
        SetDO S_8,0;
        MoveL Target_110,v2000,fine,tVacuum\WObj:=Principal;
    ENDPROC

    PROC Place_5_PPo()
        MoveL Target_110,v2000,z10,tVacuum\WObj:=Principal;
        MoveL Target_160,v300,fine,tVacuum\WObj:=Principal;
        SetDO S_8,1;
        SetDO S_8,0;
        MoveL Target_110,v2000,fine,tVacuum\WObj:=Principal;
    ENDPROC

    PROC Place_6_PPo()
        MoveL Target_110,v2000,z10,tVacuum\WObj:=Principal;
        MoveL Target_170,v300,fine,tVacuum\WObj:=Principal;
        SetDO S_8,1;
        SetDO S_8,0;
        MoveL Target_110,v2000,fine,tVacuum\WObj:=Principal;
        Home_R3;
    ENDPROC
    PROC Home()
        MoveJ Target_10,v2500,z1,tVacuum\WObj:=Plato_P;
    ENDPROC
ENDMODULE

--- Backups/Controlador_Vajilla/SYSPAR/EIO.cfg ---
EIO:CFG_1.0:6:1::
#
EIO_SIGNAL:

      -Name "S_1" -SignalType "DO" -Label "Activa Attach R1"

      -Name "S_2" -SignalType "DO" -Label "Desactiva Attach R1"

      -Name "En_1" -SignalType "DI" -Label "Sensor de línea PH"

      -Name "S_3" -SignalType "DO" -Label "Activa Conveyor principal"

      -Name "En_2" -SignalType "DI" -Label "Sensor de Plano Caja 1"

      -Name "En_3" -SignalType "DI" -Label "Sensores de linea PP y PPo"

      -Name "En_4" -SignalType "DI" -Label "Sensor de Plano Caja 2"

      -Name "S_4" -SignalType "DO" -Label "Activa Attach R3 Plato Pando"

      -Name "S_5" -SignalType "DO" -Label "Desactivar Attach R3 Plato Pando"

      -Name "S_6" -SignalType "DO" -Label "Aviso inactividad R3"

      -Name "En_5" -SignalType "DI" -Label "Entrada Inactividad R3"

      -Name "S_7" -SignalType "DO" -Label "Activa Attach R3 Plato Postre"

      -Name "S_8" -SignalType "DO" -Label "Desactivar Attach R3 Plato Postre"

      -Name "En_6" -SignalType "DI" -Label "Sensor de línea Vaso"

      -Name "S_9" -SignalType "DO" -Label "Activar Attach R2"

      -Name "S_10" -SignalType "DO" -Label "Desactivar Attach R2"
